TYPE DUT :
STRUCT
END_STRUCT
END_TYPE

(* stored: Version 1.1.0.1, ProductVersion 3.1.4024.3
   DUT DUT: Id {e4391cc7-031f-4426-908c-124e886d9f79} *)
